(* IEC 61131-3 sources: opcua/plc_code/VarMonitor, 6 files *)

(* ---- VarMonTypes.typ ---- *)
(********************************************************************
 * VarMonitor — Type definitions
 ********************************************************************)
TYPE
    VM_States_enum : (
        VM_STATE_INIT := 0,
        VM_STATE_LISTEN,
        VM_STATE_RUNNING,
        VM_STATE_ERROR
    );

    (* Type codes for the wire protocol *)
    VM_TypeCode_enum : (
        VM_TYPE_BOOL   := 0,
        VM_TYPE_INT    := 1,
        VM_TYPE_UINT   := 2,
        VM_TYPE_DINT   := 3,
        VM_TYPE_UDINT  := 4,
        VM_TYPE_REAL   := 5,
        VM_TYPE_LREAL  := 6,
        VM_TYPE_STRING := 7,
        VM_TYPE_USINT  := 8,
        VM_TYPE_SINT   := 9
    );

    (* Variable registry entry — maps ID to memory address *)
    VM_VarEntry_typ : STRUCT
        pAddress : UDINT;       (* Memory address from ADR() *)
        typeCode : USINT;       (* VM_TypeCode_enum *)
        dataSize : USINT;       (* Bytes for this type (0 for STRING = variable) *)
        name     : STRING[120]; (* Full variable path — for registry response *)
    END_STRUCT;

END_TYPE

(* ---- VarMon_ProcessCmd.st ---- *)
(********************************************************************
 * VarMon_ProcessCommand — Parse incoming TCP subscription command
 *
 * TCP Command format:
 *   [CMD:1 byte][COUNT:2 bytes LE][PAYLOAD: COUNT x 2 bytes LE]
 ********************************************************************)
ACTION VarMon_ProcessCommand:

    vmCmdByte := vmTcpRxBuf[0];
    vmCmdCount := USINT_TO_UINT(vmTcpRxBuf[1]) + USINT_TO_UINT(vmTcpRxBuf[2]) * 256;

    CASE vmCmdByte OF

        (* 0x01: SET — replace entire subscription list *)
        1:
            vmSubCount := 0;
            FOR vmIdx := 0 TO vmCmdCount - 1 DO
                IF vmIdx < VM_MAX_SUBSCRIPTIONS THEN
                    vmSubscription[vmIdx] := USINT_TO_UINT(vmTcpRxBuf[3 + vmIdx * 2]) +
                                             USINT_TO_UINT(vmTcpRxBuf[4 + vmIdx * 2]) * 256;
                    vmSubCount := vmSubCount + 1;
                END_IF;
            END_FOR;

            (* Send ACK back *)
            vmTcpTxBuf[0] := 16#01;  (* ACK *)
            vmTcpTxBuf[1] := UINT_TO_USINT(vmSubCount MOD 256);
            vmTcpTxBuf[2] := UINT_TO_USINT(vmSubCount / 256);
            vmTcpSend.enable := TRUE;
            vmTcpSend.ident := vmTcpClientIdent;
            vmTcpSend.pData := ADR(vmTcpTxBuf);
            vmTcpSend.datalen := 3;
            vmTcpSend.flags := 0;
            vmTcpSend();

        (* 0x02: ADD — add variables to subscription *)
        2:
            FOR vmIdx := 0 TO vmCmdCount - 1 DO
                IF vmSubCount < VM_MAX_SUBSCRIPTIONS THEN
                    vmSubscription[vmSubCount] :=
                        USINT_TO_UINT(vmTcpRxBuf[3 + vmIdx * 2]) +
                        USINT_TO_UINT(vmTcpRxBuf[4 + vmIdx * 2]) * 256;
                    vmSubCount := vmSubCount + 1;
                END_IF;
            END_FOR;

        (* 0x03: REMOVE — remove variables from subscription *)
        3:
            (* Simple: mark and compact *)
            FOR vmIdx := 0 TO vmCmdCount - 1 DO
                vmVarId := USINT_TO_UINT(vmTcpRxBuf[3 + vmIdx * 2]) +
                           USINT_TO_UINT(vmTcpRxBuf[4 + vmIdx * 2]) * 256;
                FOR vmIdx2 := 0 TO vmSubCount - 1 DO
                    IF vmSubscription[vmIdx2] = vmVarId THEN
                        (* Shift rest down *)
                        FOR vmIdx3 := vmIdx2 TO vmSubCount - 2 DO
                            vmSubscription[vmIdx3] := vmSubscription[vmIdx3 + 1];
                        END_FOR;
                        vmSubCount := vmSubCount - 1;
                    END_IF;
                END_FOR;
            END_FOR;

        (* 0x04: SET INTERVAL — set send rate *)
        4:
            vmSendIntervalMs := vmCmdCount;  (* Reuse count field as interval *)

        (* 0xFF: HEARTBEAT / STATUS *)
        255:
            vmTcpTxBuf[0] := 16#FF;
            vmTcpTxBuf[1] := UINT_TO_USINT(vmSubCount MOD 256);
            vmTcpTxBuf[2] := UINT_TO_USINT(vmSubCount / 256);
            vmTcpTxBuf[3] := UINT_TO_USINT(vmRegCount MOD 256);
            vmTcpTxBuf[4] := UINT_TO_USINT(vmRegCount / 256);
            vmTcpSend.enable := TRUE;
            vmTcpSend.ident := vmTcpClientIdent;
            vmTcpSend.pData := ADR(vmTcpTxBuf);
            vmTcpSend.datalen := 5;
            vmTcpSend.flags := 0;
            vmTcpSend();

    END_CASE;

END_ACTION

(* ---- VarMon_RegInit.st ---- *)
(********************************************************************
 * VarMon Registry Init — AUTO-GENERATED EXAMPLE
 *
 * This file shows how to register PLC variables with the VarMonitor.
 * In your real project, run plc_var_codegen.py to generate this
 * from plc_var_registry.json.
 *
 * Each entry maps a var_id (index) to a PLC variable's memory address.
 ********************************************************************)
ACTION VarMon_RegInit:

    vmRegCount := 0;

    (* ── Example: Exit subsystem interface ── *)

    (* gExitCtrl.In.Cmd.FullMechInit *)
    vmRegistry[0].pAddress := ADR(gExitCtrl.In.Cmd.FullMechInit);
    vmRegistry[0].typeCode := 0;  (* BOOL *)
    vmRegistry[0].dataSize := 1;
    vmRegistry[0].name := 'gExitCtrl.In.Cmd.FullMechInit';

    (* gExitCtrl.In.Cmd.Stop *)
    vmRegistry[1].pAddress := ADR(gExitCtrl.In.Cmd.Stop);
    vmRegistry[1].typeCode := 0;  (* BOOL *)
    vmRegistry[1].dataSize := 1;
    vmRegistry[1].name := 'gExitCtrl.In.Cmd.Stop';

    (* gExitCtrl.Out.Status.AtReady *)
    vmRegistry[2].pAddress := ADR(gExitCtrl.Out.Status.AtReady);
    vmRegistry[2].typeCode := 0;  (* BOOL *)
    vmRegistry[2].dataSize := 1;
    vmRegistry[2].name := 'gExitCtrl.Out.Status.AtReady';

    (* gWHS_Ctrl.Input.Cmd.Print *)
    vmRegistry[3].pAddress := ADR(gWHS_Ctrl.Input.Cmd.Print);
    vmRegistry[3].typeCode := 0;  (* BOOL *)
    vmRegistry[3].dataSize := 1;
    vmRegistry[3].name := 'gWHS_Ctrl.Input.Cmd.Print';

    (* gWHS_Ctrl.Output.Status.AtPrint *)
    vmRegistry[4].pAddress := ADR(gWHS_Ctrl.Output.Status.AtPrint);
    vmRegistry[4].typeCode := 0;  (* BOOL *)
    vmRegistry[4].dataSize := 1;
    vmRegistry[4].name := 'gWHS_Ctrl.Output.Status.AtPrint';

    (* gPrintSpeed *)
    vmRegistry[5].pAddress := ADR(gPrintSpeed);
    vmRegistry[5].typeCode := 5;  (* REAL *)
    vmRegistry[5].dataSize := 4;
    vmRegistry[5].name := 'gPrintSpeed';

    (* ... continue for all variables you want to expose ... *)
    (* Run: python plc_var_codegen.py to generate the full list *)

    vmRegCount := 6;  (* Update with actual count *)

END_ACTION

(* ---- VarMon_SendUpdate.st ---- *)
(********************************************************************
 * VarMon_SendUpdate — Pack subscribed variable values into UDP packet
 *
 * Packet format:
 *   [MAGIC:2B = 0xAB01][SEQ:4B][TIMESTAMP:4B][COUNT:2B]
 *   For each var: [VAR_ID:2B][TYPE:1B][VALUE: variable]
 ********************************************************************)
ACTION VarMon_SendUpdate:

    vmBufPos := 0;

    (* ── Header ── *)
    (* Magic *)
    vmUdpBuf[0] := 16#01;  (* Low byte of 0xAB01 *)
    vmUdpBuf[1] := 16#AB;  (* High byte *)
    vmBufPos := 2;

    (* Sequence number — 4 bytes LE *)
    brsmemcpy(ADR(vmUdpBuf[vmBufPos]), ADR(vmSeqNum), 4);
    vmBufPos := vmBufPos + 4;

    (* Timestamp — 4 bytes LE (ms since boot) *)
    vmTempUdint := clock_ms();
    brsmemcpy(ADR(vmUdpBuf[vmBufPos]), ADR(vmTempUdint), 4);
    vmBufPos := vmBufPos + 4;

    (* Count placeholder — fill after packing *)
    vmCountPos := vmBufPos;
    vmBufPos := vmBufPos + 2;

    (* ── Pack each subscribed variable ── *)
    vmPackedCount := 0;

    FOR vmIdx := 0 TO vmSubCount - 1 DO
        vmVarId := vmSubscription[vmIdx];

        (* Bounds check *)
        IF vmVarId >= vmRegCount THEN
            (* Skip invalid var_id *)
            (* Continue loop *)
        ELSIF vmBufPos > (VM_UDP_BUF_SIZE - 12) THEN
            (* Buffer nearly full — send what we have, rest in next packet *)
            (* Exit loop *)
            EXIT;
        ELSE
            (* Pack var_id — 2 bytes LE *)
            vmUdpBuf[vmBufPos] := UINT_TO_USINT(vmVarId MOD 256);
            vmUdpBuf[vmBufPos + 1] := UINT_TO_USINT(vmVarId / 256);
            vmBufPos := vmBufPos + 2;

            (* Pack type code — 1 byte *)
            vmUdpBuf[vmBufPos] := vmRegistry[vmVarId].typeCode;
            vmBufPos := vmBufPos + 1;

            (* Pack value based on type *)
            CASE vmRegistry[vmVarId].typeCode OF

                0: (* BOOL — 1 byte *)
                    brsmemcpy(ADR(vmTempBool), vmRegistry[vmVarId].pAddress, 1);
                    IF vmTempBool THEN
                        vmUdpBuf[vmBufPos] := 1;
                    ELSE
                        vmUdpBuf[vmBufPos] := 0;
                    END_IF;
                    vmBufPos := vmBufPos + 1;

                1: (* INT — 2 bytes LE *)
                    brsmemcpy(ADR(vmUdpBuf[vmBufPos]), vmRegistry[vmVarId].pAddress, 2);
                    vmBufPos := vmBufPos + 2;

                2: (* UINT — 2 bytes LE *)
                    brsmemcpy(ADR(vmUdpBuf[vmBufPos]), vmRegistry[vmVarId].pAddress, 2);
                    vmBufPos := vmBufPos + 2;

                3: (* DINT — 4 bytes LE *)
                    brsmemcpy(ADR(vmUdpBuf[vmBufPos]), vmRegistry[vmVarId].pAddress, 4);
                    vmBufPos := vmBufPos + 4;

                4: (* UDINT — 4 bytes LE *)
                    brsmemcpy(ADR(vmUdpBuf[vmBufPos]), vmRegistry[vmVarId].pAddress, 4);
                    vmBufPos := vmBufPos + 4;

                5: (* REAL — 4 bytes LE (IEEE 754) *)
                    brsmemcpy(ADR(vmUdpBuf[vmBufPos]), vmRegistry[vmVarId].pAddress, 4);
                    vmBufPos := vmBufPos + 4;

                6: (* LREAL — 8 bytes LE *)
                    brsmemcpy(ADR(vmUdpBuf[vmBufPos]), vmRegistry[vmVarId].pAddress, 8);
                    vmBufPos := vmBufPos + 8;

                7: (* STRING — 1 byte length + chars *)
                    brsmemcpy(ADR(vmTempString), vmRegistry[vmVarId].pAddress, 81);
                    vmTempStrLen := UDINT_TO_USINT(brsstrlen(ADR(vmTempString)));
                    IF vmTempStrLen > 80 THEN
                        vmTempStrLen := 80;
                    END_IF;
                    vmUdpBuf[vmBufPos] := vmTempStrLen;
                    vmBufPos := vmBufPos + 1;
                    brsmemcpy(ADR(vmUdpBuf[vmBufPos]), ADR(vmTempString), vmTempStrLen);
                    vmBufPos := vmBufPos + vmTempStrLen;

                8: (* USINT — 1 byte *)
                    brsmemcpy(ADR(vmUdpBuf[vmBufPos]), vmRegistry[vmVarId].pAddress, 1);
                    vmBufPos := vmBufPos + 1;

                9: (* SINT — 1 byte *)
                    brsmemcpy(ADR(vmUdpBuf[vmBufPos]), vmRegistry[vmVarId].pAddress, 1);
                    vmBufPos := vmBufPos + 1;

            END_CASE;

            vmPackedCount := vmPackedCount + 1;
        END_IF;
    END_FOR;

    (* Fill in the count field *)
    vmUdpBuf[vmCountPos] := UINT_TO_USINT(vmPackedCount MOD 256);
    vmUdpBuf[vmCountPos + 1] := UINT_TO_USINT(vmPackedCount / 256);

    (* ── Send UDP packet ── *)
    vmUdpSend.enable := TRUE;
    vmUdpSend.ident := vmUdpIdent;
    vmUdpSend.pHost := ADR(vmClientIpAddr);
    vmUdpSend.port := vmClientPort;
    vmUdpSend.pData := ADR(vmUdpBuf);
    vmUdpSend.datalen := vmBufPos;
    vmUdpSend.flags := 0;
    vmUdpSend();

    vmSeqNum := vmSeqNum + 1;

END_ACTION

(* ---- VarMonCyclic.st ---- *)
(********************************************************************
 * VarMonitor — Variable monitoring via UDP/TCP
 *
 * Architecture:
 *   - TCP server (port 55000): receives subscription commands
 *   - UDP sender (port 55001): sends variable values to subscriber
 *
 * Protocol:
 *   TCP Command format (from Python):
 *     [CMD:1 byte][COUNT:2 bytes LE][VAR_IDs: COUNT x 2 bytes LE]
 *     CMD = 0x01: SET subscription (replace all)
 *     CMD = 0x02: ADD to subscription
 *     CMD = 0x03: REMOVE from subscription
 *     CMD = 0x04: SET interval (COUNT=interval_ms as UINT)
 *     CMD = 0xFF: Request heartbeat/status
 *
 *   UDP Packet format (to Python):
 *     [MAGIC:2 bytes = 0xAB01]
 *     [SEQ:4 bytes UDINT]
 *     [TIMESTAMP:4 bytes UDINT (ms since boot)]
 *     [COUNT:2 bytes UINT - number of variables]
 *     For each variable:
 *       [VAR_ID:2 bytes UINT]
 *       [TYPE:1 byte (0=BOOL,1=INT,2=UINT,3=DINT,4=UDINT,5=REAL,6=LREAL,7=STRING)]
 *       [VALUE: variable length based on type]
 *         BOOL: 1 byte
 *         INT/UINT: 2 bytes LE
 *         DINT/UDINT: 4 bytes LE
 *         REAL: 4 bytes LE (IEEE 754)
 *         LREAL: 8 bytes LE (IEEE 754)
 *         STRING: 1 byte length + N bytes chars
 ********************************************************************)

PROGRAM _INIT
    (* TCP Server setup *)
    vmTcpOpen.enable := TRUE;
    vmTcpOpen.pIfAddr := 0;           (* All interfaces *)
    vmTcpOpen.port := VM_TCP_PORT;
    vmTcpOpen.options := 0;

    (* UDP setup *)
    vmUdpOpen.enable := TRUE;
    vmUdpOpen.pIfAddr := 0;
    vmUdpOpen.port := 0;              (* Any local port for sending *)
    vmUdpOpen.options := 0;

    vmState := VM_STATE_INIT;
    vmSeqNum := 0;
    vmSubCount := 0;
    vmSendIntervalMs := 10;           (* Default 10ms send interval *)
    vmClientConnected := FALSE;
    vmClientPort := VM_UDP_PORT;
    vmLastSendTime := 0;

    (* Clear subscription list *)
    FOR vmIdx := 0 TO VM_MAX_SUBSCRIPTIONS - 1 DO
        vmSubscription[vmIdx] := 0;
    END_FOR;

    (* Initialize variable registry —
       This maps var_id (index) to actual PLC variable addresses.
       Generated by plc_var_scanner.py — see VarMonReg_Init *)
END_PROGRAM

PROGRAM _CYCLIC
    CASE vmState OF

        (* ─── INIT: Open TCP + UDP sockets ─── *)
        VM_STATE_INIT:
            vmTcpOpen();
            vmUdpOpen();

            IF vmTcpOpen.status = 0 AND vmUdpOpen.status = 0 THEN
                vmTcpIdent := vmTcpOpen.ident;
                vmUdpIdent := vmUdpOpen.ident;

                (* Start TCP server listening *)
                vmTcpServer.enable := TRUE;
                vmTcpServer.ident := vmTcpIdent;
                vmTcpServer.backlog := 1;
                vmTcpServer.pIpAddr := ADR(vmClientIpAddr);

                vmState := VM_STATE_LISTEN;
            ELSIF vmTcpOpen.status <> ERR_FUB_BUSY AND
                  vmUdpOpen.status <> ERR_FUB_BUSY THEN
                (* Error — retry after delay *)
                vmState := VM_STATE_ERROR;
            END_IF;

        (* ─── LISTEN: Wait for TCP client connection ─── *)
        VM_STATE_LISTEN:
            vmTcpServer();

            IF vmTcpServer.status = 0 THEN
                vmTcpClientIdent := vmTcpServer.identclnt;
                vmClientConnected := TRUE;
                vmState := VM_STATE_RUNNING;

                (* Setup TCP receive *)
                vmTcpRecv.enable := TRUE;
                vmTcpRecv.ident := vmTcpClientIdent;
                vmTcpRecv.pData := ADR(vmTcpRxBuf);
                vmTcpRecv.datamax := SIZEOF(vmTcpRxBuf);
                vmTcpRecv.flags := 0;
            ELSIF vmTcpServer.status <> ERR_FUB_BUSY THEN
                vmState := VM_STATE_ERROR;
            END_IF;

        (* ─── RUNNING: Process commands + send data ─── *)
        VM_STATE_RUNNING:
            (* Check for incoming TCP commands *)
            vmTcpRecv();

            IF vmTcpRecv.status = 0 THEN
                (* Process received command *)
                IF vmTcpRecv.recvlen > 0 THEN
                    VarMon_ProcessCommand();
                END_IF;
            ELSIF vmTcpRecv.status = tcpERR_NOT_CONNECTED THEN
                (* Client disconnected *)
                vmClientConnected := FALSE;
                vmSubCount := 0;
                vmState := VM_STATE_LISTEN;
            END_IF;

            (* Send subscribed variable values via UDP *)
            IF vmClientConnected AND vmSubCount > 0 THEN
                clock_ms := clock_ms();
                IF (clock_ms - vmLastSendTime) >= vmSendIntervalMs THEN
                    VarMon_SendUpdate();
                    vmLastSendTime := clock_ms;
                END_IF;
            END_IF;

        (* ─── ERROR: Handle errors ─── *)
        VM_STATE_ERROR:
            (* Close and restart *)
            vmTcpClose.enable := TRUE;
            vmTcpClose.ident := vmTcpIdent;
            vmTcpClose();
            vmUdpClose.enable := TRUE;
            vmUdpClose.ident := vmUdpIdent;
            vmUdpClose();

            IF vmTcpClose.status <> ERR_FUB_BUSY AND
               vmUdpClose.status <> ERR_FUB_BUSY THEN
                vmState := VM_STATE_INIT;
            END_IF;

    END_CASE;
END_PROGRAM

PROGRAM _EXIT
    vmTcpClose.enable := TRUE;
    vmTcpClose.ident := vmTcpIdent;
    vmTcpClose.how := 0;
    vmTcpClose();

    vmUdpClose.enable := TRUE;
    vmUdpClose.ident := vmUdpIdent;
    vmUdpClose();
END_PROGRAM

(* ---- VarMonVars.var ---- *)
(********************************************************************
 * VarMonitor — Variable declarations
 ********************************************************************)
VAR CONSTANT
    VM_TCP_PORT : UINT := 55000;        (* TCP command port *)
    VM_UDP_PORT : UINT := 55001;        (* UDP data port on Python side *)
    VM_MAX_SUBSCRIPTIONS : UINT := 500; (* Max variables to subscribe *)
    VM_MAX_REGISTRY : UINT := 2000;     (* Max variables in registry *)
    VM_UDP_BUF_SIZE : UINT := 1400;     (* Max UDP packet size *)
    VM_TCP_BUF_SIZE : UINT := 2048;     (* TCP receive buffer *)
    VM_MAGIC : UINT := 16#AB01;         (* Packet magic number *)
END_VAR

VAR
    (* State machine *)
    vmState : VM_States_enum;
    vmIdx   : UINT;

    (* TCP server *)
    vmTcpOpen    : TcpOpen;
    vmTcpServer  : TcpServer;
    vmTcpRecv    : TcpRecv;
    vmTcpSend    : TcpSend;
    vmTcpClose   : TcpClose;
    vmTcpIdent   : UDINT;
    vmTcpClientIdent : UDINT;
    vmTcpRxBuf   : ARRAY[0..2047] OF USINT;
    vmTcpTxBuf   : ARRAY[0..2047] OF USINT;
    vmClientIpAddr : STRING[20];
    vmClientConnected : BOOL;

    (* UDP sender *)
    vmUdpOpen    : UdpOpen;
    vmUdpSend    : UdpSend;
    vmUdpClose   : UdpClose;
    vmUdpIdent   : UDINT;
    vmUdpBuf     : ARRAY[0..1399] OF USINT;  (* Send buffer *)
    vmClientPort : UINT;

    (* Subscription management *)
    vmSubscription : ARRAY[0..499] OF UINT;  (* Active var_id list *)
    vmSubCount   : UINT;                      (* Number of active subscriptions *)
    vmSendIntervalMs : UINT;                  (* Send interval in ms *)
    vmSeqNum     : UDINT;                     (* Packet sequence counter *)
    vmLastSendTime : UDINT;                   (* Last send timestamp *)

    (* Variable registry — populated in _INIT or by code generator *)
    vmRegistry   : ARRAY[0..1999] OF VM_VarEntry_typ;
    vmRegCount   : UINT;                      (* Number of registered variables *)

    (* Temp vars for packing *)
    vmBufPos     : UINT;
    vmTempBool   : BOOL;
    vmTempInt    : INT;
    vmTempUint   : UINT;
    vmTempDint   : DINT;
    vmTempUdint  : UDINT;
    vmTempReal   : REAL;
    vmTempLreal  : LREAL;
    vmTempUsint  : USINT;
    vmTempString : STRING[80];
    vmTempStrLen : USINT;
    vmVarId      : UINT;
END_VAR
